FUNCTION_BLOCK FB_PrePalletizer EXTENDS FB_Chain
VAR_INPUT
END_VAR
VAR_OUTPUT
END_VAR
VAR
END_VAR

END_FUNCTION_BLOCK

(* stored: Version 1.1.0.1, ProductVersion 3.1.4024.0
   POU FB_PrePalletizer: Id {5dff49bc-e989-4c97-b519-5d232efdac58}, SpecialFunc None *)
